// TIA Portal V17 export
// export: Created 2026-04-13T11:12:53.2012406Z, ExportSetting WithDefaults, DisplayName Totally Integrated Automation Portal, DisplayVersion V17 Update 4, DisplayName TIA Portal Openness, DisplayVersion V17 Update 4, DisplayName TIA Portal Version Control Interface, DisplayVersion V17, DisplayName SINAMICS Startdrive Advanced, DisplayVersion V17, DisplayName SINAMICS Startdrive G130, G150, S120, S150, SINAMICS MV, S210, DisplayVersion V17, DisplayName SINAMICS Startdrive G110M, G120, G120C, G120D, G120P, G115D, DisplayVersion V17, DisplayName STEP 7 Professional, DisplayVersion V17 Update 4, DisplayName STEP 7 Safety, DisplayVersion V17, DisplayName WinCC Professional, DisplayVersion V17 Update 4
TagTable "KS"
  KS_JF进风流量上阈值 : Real  (PLC tag KS.JF进风流量上阈值, HMI_连接_1, 1 s)
  KS_JF进风流量下阈值 : Real  (PLC tag KS.JF进风流量下阈值, HMI_连接_1, 1 s)
  KS_ZT主塔压力引风升临界 : Real  (PLC tag KS.ZT主塔压力引风升临界, HMI_连接_1, 1 s)
  KS_JF进风流量引风关临界 : Real  (PLC tag KS.JF进风流量引风关临界, HMI_连接_1, 1 s)
  KS_JF进风流量送风关临界 : Real  (PLC tag KS.JF进风流量送风关临界, HMI_连接_1, 1 s)
  KS_SF送风机1分钟升速 : Real  (PLC tag KS.SF送风机1分钟升速, HMI_连接_1, 1 s)
  KS_YP预喷雾检测主塔压力维持时间 : Int  (PLC tag KS.YP预喷雾检测主塔压力维持时间, HMI_连接_1, 1 s)
  KS_YP预喷雾检测高压 : Real  (PLC tag KS.YP预喷雾检测高压, HMI_连接_1, 1 s)
  KS_YP预喷雾检测低压 : Real  (PLC tag KS.YP预喷雾检测低压, HMI_连接_1, 1 s)
  KS_YP预喷雾检测系统结果 : Int  (PLC tag KS.YP预喷雾检测系统结果, HMI_连接_1, 1 s)
  KS_YP预喷雾检测系统正常 : Bool  (PLC tag KS.YP预喷雾检测系统正常, HMI_连接_1, 1 s)
  KS_YP预喷雾进风流量 : Real  (PLC tag KS.YP预喷雾进风流量, HMI_连接_1, 1 s)
  KS_YP预喷雾-离雾-进温 : Real  (PLC tag KS.YP预喷雾-离雾-进温, HMI_连接_1, 1 s)
  KS_YP预喷雾-离雾-出温 : Real  (PLC tag KS.YP预喷雾-离雾-出温, HMI_连接_1, 1 s)
  KS_YP预喷雾温稳正式时间 : Int  (PLC tag KS.YP预喷雾温稳正式时间, HMI_连接_1, 1 s)
  KS_GJ关机洗喷头时间 : Int  (PLC tag KS.GJ关机洗喷头时间, HMI_连接_1, 1 s)
  KS_GJ关机-停水-出温 : Real  (PLC tag KS.GJ关机-停水-出温, HMI_连接_1, 1 s)
  KS_GJ关机-停水-停雾 : DInt  (PLC tag KS.GJ关机-停水-停雾, HMI_连接_1, 1 s)
  KS_GJ关机-四参数关-进温 : Real  (PLC tag KS.GJ关机-四参数关-进温, HMI_连接_1, 1 s)
  KS_GJ关机-输送-送温 : Real  (PLC tag KS.GJ关机-输送-送温, HMI_连接_1, 1 s)
  KS_ZD自动运行报警 : Bool  (PLC tag KS.ZD自动运行报警, HMI_连接_1, 1 s)
  KS_BD步段运行_秒 : Int  (PLC tag KS.BD步段运行_秒, HMI_连接_1, 1 s)
  KS_BD步段运行_分 : Int  (PLC tag KS.BD步段运行_分, HMI_连接_1, 1 s)
  KS_BD步段运行_时 : Int  (PLC tag KS.BD步段运行_时, HMI_连接_1, 1 s)
  KS_ZY总运行_秒 : Int  (PLC tag KS.ZY总运行_秒, HMI_连接_1, 1 s)
  KS_ZY总运行_分 : Int  (PLC tag KS.ZY总运行_分, HMI_连接_1, 1 s)
  KS_ZY总运行_时 : Int  (PLC tag KS.ZY总运行_时, HMI_连接_1, 1 s)
  KS_JL进料_时 : Int  (PLC tag KS.JL进料_时, HMI_连接_1, 1 s)
  KS_JL进料_分 : Int  (PLC tag KS.JL进料_分, HMI_连接_1, 1 s)
  KS_JL进料_秒 : Int  (PLC tag KS.JL进料_秒, HMI_连接_1, 1 s)
  KS_BD步段设定 : Int  (PLC tag KS.BD步段设定, HMI_连接_1, 1 s)
  KS_BD步段运行 : Int  (PLC tag KS.BD步段运行, HMI_连接_1, 1 s)
  KS_ZD自动停止 : Bool  (PLC tag KS.ZD自动停止, HMI_连接_1, 1 s)
  KS_AQ安全停机 : Bool  (PLC tag KS.AQ安全停机, HMI_连接_1, 1 s)
  KS_JL进料时间设定 : Real  (PLC tag KS.JL进料时间设定, HMI_连接_1, 1 s)
  KS_XT系统状态 : Int  (PLC tag KS.XT系统状态, HMI_连接_1, 1 s)
  KS_JL进料进风阈值 : Real  (PLC tag KS.JL进料进风阈值, HMI_连接_1, 1 s)
  KS_JL进料出风条件 : Real  (PLC tag KS.JL进料出风条件, HMI_连接_1, 1 s)
  KS_CF出温高报 : Real  (PLC tag KS.CF出温高报, HMI_连接_1, 1 s)
  KS_CF出温高高报 : Real  (PLC tag KS.CF出温高高报, HMI_连接_1, 1 s)
  KS_WQ尾温高报 : Real  (PLC tag KS.WQ尾温高报, HMI_连接_1, 1 s)
  KS_WQ尾温高高报 : Real  (PLC tag KS.WQ尾温高高报, HMI_连接_1, 1 s)
  KS_JF进温高报 : Real  (PLC tag KS.JF进温高报, HMI_连接_1, 1 s)
  KS_JF进温高高报 : Real  (PLC tag KS.JF进温高高报, HMI_连接_1, 1 s)
